// TwinCAT 3 PLC project PLC
// ProgramVersion: 3.1.4026.19
// CompilerDefines: VISU_USEPROPERTYINFO
// libraries:
//   Tc2_Standard, * (Beckhoff Automation GmbH)
//   Tc2_System, * (Beckhoff Automation GmbH)
// project tree:
//   / GlobalTextList.TcGTLO, PlcTask.TcTTO, Visualization Manager.TcVMO (not stored)
//   POUs/ MAIN.TcPOU
//   VISUs/ Visualization.TcVIS

CONFIGURATION PLC
    RESOURCE PLC ON TwinCAT3
        TASK PlcTask(INTERVAL := T#10ms, PRIORITY := 20);
        PROGRAM MAIN WITH PlcTask : MAIN;
    END_RESOURCE
END_CONFIGURATION

// ---- POUs/MAIN.TcPOU
PROGRAM MAIN
VAR
	nRawAnalogInput : INT;
	fMotorSpeedPercent: REAL;
END_VAR

IF nRawAnalogInput < 0 THEN
	nRawAnalogInput :=0;
	
ELSIF nRawAnalogInput > 32767 THEN
	nRawAnalogInput := 32767;
END_IF

fMotorSpeedPercent := (INT_TO_REAL(nRawAnalogInput)/32767.0)*100.0;

END_PROGRAM

// ---- VISUs/Visualization.TcVIS
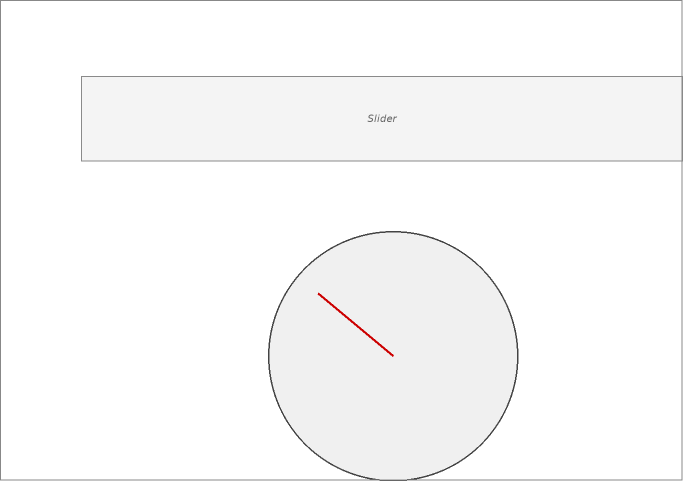
VISUALIZATION Visualization  // 683x481
    Slider (81,76 602x85), variable: MAIN.nRawAnalogInput, scale 0..32767
    Meter360 (268,231 250x250), value: MAIN.fMotorSpeedPercent, style: Meter-Meter360-Gray, scale format: %.1f, scale 0..100
END_VISUALIZATION
